INTERFACE I_NciChannelBase EXTENDS I_ComponentBase

METHOD BuildGroup
END_METHOD

PROPERTY ChannelError : BOOL
GET
END_GET
END_PROPERTY

PROPERTY ChannelErrorId : UDINT
GET
END_GET
END_PROPERTY

PROPERTY IsGrouped : BOOL
GET
END_GET
END_PROPERTY

PROPERTY IsReady : BOOL
GET
END_GET
END_PROPERTY

METHOD ResetChannel
VAR_INPUT
END_VAR
END_METHOD

METHOD Stop
VAR_INPUT
END_VAR
END_METHOD

METHOD Ungroup
VAR_INPUT
END_VAR
END_METHOD

END_INTERFACE

(* stored: Version 1.1.0.1, ProductVersion 3.1.4024.15
   Itf I_NciChannelBase: Id {621d396d-a712-4314-9317-18e0a12884ff}
   Method BuildGroup: Id {5439cb1a-b8ef-46bc-8b6a-64a9cf8db48f}
   Property ChannelError: Id {bd1a5da7-6046-4778-9051-4ddb2e401168}
   Get Get: Id {a697e5cf-f209-4696-a4b9-cdb3ab0a03f5}
   Property ChannelErrorId: Id {70652d02-87ca-4140-a719-653c0d561a22}
   Get Get: Id {3ea1bc4d-3aa1-488b-8197-01b768b74b98}
   Property IsGrouped: Id {491dcdd1-0461-4e2f-93ad-e950495e0c5b}
   Get Get: Id {2a0672f3-3a00-42b6-9201-90e777c0b9ef}
   Property IsReady: Id {6978e012-72a4-46fd-9420-9e08db683d11}
   Get Get: Id {20f89dbc-3283-43bf-b065-ce61067d03df}
   Method ResetChannel: Id {7d258806-166e-4393-948c-0dd169c6ac1a}
   Method Stop: Id {b90f03ae-c194-4529-8014-173f40a894e9}
   Method Ungroup: Id {49d61b60-7e7e-4601-a87f-20dcda08eb54} *)
